ABB RobotStudio station: GoFa_CRB15000.rsstn

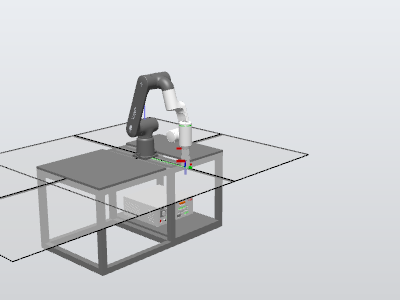
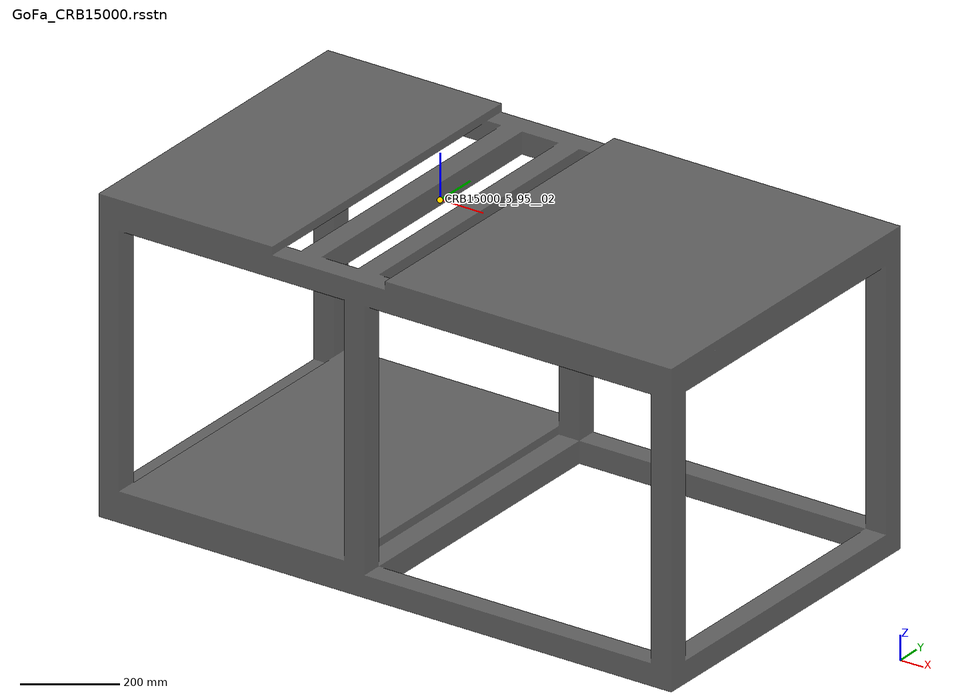
[picture v1: parts stored in the station drawn from their meshes, with robot base, taught points and paths (robot models come from the ABB library and are not in the file)]
Station Station (saved by RobotStudio 22.3.10141.1)
Controller VIRTUAL_CTRL_15000-100072
  mechanical unit ROB_1: CRB15000_5_95__02, 6 joints, base frame (0, 0, 0) mm
Layout (positions relative to the parent item):
  - controller [part, from %ABB.RobotStudio.Models.OmniCore%\OmniCore_C30.rslib] at (0, 150, -631) mm, rotated rx 0 ry 0 rz 180 deg
  - worktable [part], size 1400 x 800 x 719 mm
  - CRB15000_5_95__02 [mechanism, from Robots\CRB15000_5_95__02.rslib] at (0, 0, 0) mm; joint values [1.5708, 0.3526, 0.9141, 0, 0.3042, -0.7849] (rad or m)
  - t_measurement [mechanism, from Libraries\t_measurement.rslib] at (0, 0, 0) mm
  - t_sgraffito [mechanism, from Libraries\t_sgraffito.rslib] at (0, 0, 0) mm
  - t_gripper [mechanism, from Libraries\t_gripper.rslib] at (0.01, 478.99, 165.15) mm, rotated rx 179.99 ry -0.01 rz -45.03 deg
  - gripper [frame] at (0, 0, 150) mm, rotated rx 0 ry 0 rz 135 deg
Attachment: t_gripper is attached to CRB15000_5_95__02 / Link6
Station signals: DI ABB_Scalable_IO_0_DO16
Targets, tools, work objects and paths stored in the station, written as RAPID:
! task T_ROB1
MODULE RRC_Main
  PROC main()
  ENDPROC
ENDMODULE

! task T_ROB1
MODULE RRC_Main
  PROC main()
    r_RRC_Main;
  ENDPROC
ENDMODULE

! task T_ROB1
MODULE RRC_Base_DataTask_Rob
  TASK PERS tooldata t_RRC_Act:=[TRUE,[[0.84733,0,105],[1,0,0,0]],[0.001,[0,0,0.001],[1,0,0,0],0,0,0]];
  VAR signaldo do_RRC_Act;
  VAR signalao ao_RRC_Act;
  TASK PERS num n_RRC_Time:=1;
  VAR signalgo go_RRC_Act;
  TASK PERS speeddata v_RRC_Act:=[39,500,5000,1000];
  TASK PERS zonedata z_RRC_Act:=[TRUE,0,0,0,0,0,0];
ENDMODULE

! task T_ROB1
MODULE GOFA_ASI_Procedures
  PROC ASI_Routine2()
  ENDPROC
  PROC ASI_Routine1()
  ENDPROC
ENDMODULE

! task T_ROB1
MODULE RRC_Base_Feedback_Rob
  PROC r_RRC_FError()
  ENDPROC
  PROC r_RRC_FDone()
  ENDPROC
ENDMODULE

! task T_ROB1
MODULE RRC_Base_Instructions_Rob
  PROC r_RRC_PrintText()
    r_RRC_FDone;
    r_RRC_FError;
  ENDPROC
  PROC r_RRC_GetRobtarget()
    r_RRC_FDone;
    r_RRC_FError;
  ENDPROC
  PROC r_RRC_SetMaxSpeed()
    r_RRC_FDone;
    r_RRC_FError;
  ENDPROC
  PROC r_RRC_SetWorkObject()
    r_RRC_FDone;
    r_RRC_FError;
  ENDPROC
  PROC r_RRC_StartWatch()
    r_RRC_FDone;
    r_RRC_FError;
  ENDPROC
  PROC r_RRC_StopWatch()
    r_RRC_FDone;
    r_RRC_FDone;
    r_RRC_FError;
  ENDPROC
  PROC r_RRC_ReadWatch()
    r_RRC_FDone;
    r_RRC_FError;
  ENDPROC
  PROC r_RRC_SetDigital()
    SetDO do_RRC_Act,bm_RRC_RecBufferRob{n_RRC_ChaNr,n_RRC_ReadPtrRecBuf}.Data.V1;
    r_RRC_FDone;
    r_RRC_FError;
  ENDPROC
  PROC r_RRC_PulseDigital()
    PulseDO \High\PLength:=bm_RRC_RecBufferRob{n_RRC_ChaNr,n_RRC_ReadPtrRecBuf}.Data.V1,do_RRC_Act;
    r_RRC_FDone;
    r_RRC_FError;
  ENDPROC
  PROC r_RRC_ReadDigital()
    r_RRC_FDone;
    r_RRC_FError;
  ENDPROC
  PROC r_RRC_SetAnalog()
    SetAO ao_RRC_Act,bm_RRC_RecBufferRob{n_RRC_ChaNr,n_RRC_ReadPtrRecBuf}.Data.V1;
    r_RRC_FDone;
    r_RRC_FError;
  ENDPROC
  PROC r_RRC_ReadAnalog()
    r_RRC_FDone;
    r_RRC_FError;
  ENDPROC
  PROC r_RRC_WaitTime()
    WaitTime n_RRC_Time;
    r_RRC_FDone;
    r_RRC_FError;
  ENDPROC
  PROC r_RRC_SetGroup()
    SetGO go_RRC_Act,bm_RRC_RecBufferRob{n_RRC_ChaNr,n_RRC_ReadPtrRecBuf}.Data.V1;
    r_RRC_FDone;
    r_RRC_FError;
  ENDPROC
  PROC r_RRC_ReadGroup()
    r_RRC_FDone;
    r_RRC_FError;
  ENDPROC
  PROC r_RRC_MoveToJoints()
    r_RRC_RasJointtarget;
    r_RRC_FDone;
    r_RRC_FError;
  ENDPROC
  PROC r_RRC_GetJoints()
    r_RRC_FDone;
    r_RRC_FError;
  ENDPROC
  PROC r_RRC_MoveTo()
    ConfL \Off;
    ConfL \On;
    ConfJ \Off;
    ConfJ \On;
    r_RRC_FDone;
    r_RRC_FError;
  ENDPROC
  PROC r_RRC_Stop()
    r_RRC_FDone;
    r_RRC_FError;
  ENDPROC
  PROC r_RRC_Noop()
    r_RRC_FDone;
    r_RRC_FError;
  ENDPROC
  PROC r_RRC_SetAcceleration()
    r_RRC_FDone;
    r_RRC_FError;
  ENDPROC
  PROC r_RRC_CustomInstruction()
    r_RRC_FDone;
    r_RRC_FError;
  ENDPROC
  PROC r_RRC_SetTool()
    r_RRC_FDone;
    r_RRC_FError;
  ENDPROC
ENDMODULE

! task T_ROB1
MODULE RRC_Base_Utilities_Rob
  PROC r_RRC_RasJointtarget()
  ENDPROC
ENDMODULE

! task T_ROB1
MODULE RRC_Control_Rob
  PROC r_RRC_Main()
    WaitTime n_RRC_TimeTaskLiAll;
    WaitSyncTask id_RRC_MainSta,tl_RRC_All;
    r_RRC_InitCell;
    r_RRC_ExeJobFrmRecBuf;
    WaitSyncTask id_RRC_MainEnd,tl_RRC_All;
  ENDPROC
  PROC r_RRC_InitVar()
    r_RRC_ProgError;
  ENDPROC
  PROC r_RRC_InitCell()
    WaitSyncTask id_RRC_InitSta,tl_RRC_All;
    WaitSyncTask id_RRC_InitCtrl,tl_RRC_All;
    r_RRC_InitVar;
    WaitSyncTask id_RRC_InitEnd,tl_RRC_All;
  ENDPROC
  PROC r_RRC_ExeJobFrmRecBuf()
  ENDPROC
  PROC r_RRC_ProgError()
  ENDPROC
ENDMODULE

! task T_ROB1
MODULE RRC_Helper_Rob
  PROC r_RRC_StoJoPosInArry()
  ENDPROC
  PROC r_RRC_ExeJoPosFromArry()
    MoveAbsJ jp_RRC_Arry{n_RRC_ArryPointer},vmax,z200,tool0;
  ENDPROC
ENDMODULE

! task T_ROB1
MODULE TorqueSensorCalib
  PROC TorqueSensorCal()
  ENDPROC
ENDMODULE

! task T_ROB1
MODULE RRC_DataGlobal
  PERS num n_RRC_TimeTaskLiAll;
  VAR syncident id_RRC_MainSta;
  PERS tasks tl_RRC_All{7};
  VAR syncident id_RRC_MainEnd;
  VAR syncident id_RRC_InitSta;
  VAR syncident id_RRC_InitCtrl;
  VAR syncident id_RRC_InitEnd;
ENDMODULE

! task T_ROB1
MODULE CalibData
  PERS tooldata t_sgraffito:=[TRUE,[[0.847,0,105],[1,0,0,0]],[1,[0,0,1],[1,0,0,0],0,0,0]];
  PERS tooldata t_measurement:=[TRUE,[[0,0,109],[1,0,0,0]],[1,[0,0,1],[1,0,0,0],0,0,0]];
  PERS tooldata t_gripper:=[TRUE,[[0,0,150],[0.382683432,0,0,0.923879533]],[1,[0,0,1],[1,0,0,0],0,0,0]];
ENDMODULE

